FUNCTION_BLOCK AOI_LoadWoodBunk
VAR_INPUT
	execute : BOOL;
END_VAR
VAR_IN_OUT CONSTANT
	sectionID : SectionEnum;
END_VAR
VAR_IN_OUT
	robot : RobotA21;
	table : StagingTable;
	suctions : ARRAY[*] OF SuctionPad;
	//if assigned using . operator instead of (), this becomes a pointer - use numPads isntead of UPPER_BOUND/LOWER_BOUND
	loadedMaterials : ARRAY[*] OF STRING;
END_VAR
VAR_INPUT
	surfaceID : Surface;
	material : STRING;
	
	//suctionI1 : DINT;
	//suctionI2 : DINT;
	
	numPads : DINT;
END_VAR
VAR_OUTPUT
	busy : BOOL;
	done : BOOL;
	error : BOOL;
	
	recovery : BOOL;
	failCounter : INT;
	
	donePulse : BOOL;
END_VAR
VAR
	run : BOOL;
	trigger : R_TRIG;
	doneTrigger : R_TRIG;
	
	slot : INT;
	
	suctionTimer : TON;
	step : (IDLE, PREP_ROBOT, GET_FROM_TABLE, LOAD_TO_INSERTION, COMPLETE, RECOVERY_IDLE, RECOVERY_REMOVE, RECOVERY_STAGE);
END_VAR
VAR
	start, end : DINT;
	i : DINT;
	test : BOOL;
END_VAR
VAR_STAT CONSTANT
	suctionDelay : TIME := T#2S;
	suctionDistance : INT := 10;
END_VAR

{warning disable C0371}
(*
IF suctions <> 0 THEN
	FOR i:=0 TO numPads-1 BY 1 DO
		suctions[i].enable := test;
	END_FOR
END_IF
*)
trigger(CLK:= execute, Q=> );
doneTrigger(CLK:= done, Q=> donePulse);
busy := trigger.Q OR step > 0;

IF step > IDLE AND_THEN NOT preExecution() THEN //conditions to track before execution
	RETURN;
END_IF

(*
if required bunk was not found on table - restage entire table
if bunk was not loaded correctly - remove bunk, then restage entire table
*)

start := LOWER_BOUND(loadedMaterials, 1);
end := UPPER_BOUND(loadedMaterials, 1);

CASE step OF
	IDLE:
		IF trigger.Q THEN //reset outputs
			done := FALSE;
			error := FALSE;
			recovery := FALSE;
			
			step := PREP_ROBOT;
		END_IF
		
	PREP_ROBOT:
		robot.clearCommand();
		IF robot.Ready THEN
			step := GET_FROM_TABLE;
			slot := 0;
		END_IF
		
	GET_FROM_TABLE:		
		IF slot < 1 AND_THEN NOT table.findSlot(material := material, index => slot) THEN
			step := RECOVERY_STAGE;
			RETURN;
		END_IF
		
		IF NOT table.isOccupied(i := slot) AND table.getSlot(i := slot) <> '' THEN //move from table to robot gripper
			robot.HoldMaterial := table.getSlot(i := slot);
			table.remove(i := slot, material => );
		END_IF
		
		IF robot.Done THEN
			step := COMPLETE;
			RETURN;
		ELSIF robot.materialAtHoldingPosition >= 1 AND robot.materialAtHoldingPosition <= 8 THEN
			step := LOAD_TO_INSERTION;
			RETURN;
		END_IF
		
		CASE surfaceID OF
			Surface.TOP: 					robot.setGroup(group := 1, value := A21.LOAD_BUNK_TOP); 
			Surface.LEFT, Surface.RIGHT: 	robot.setGroup(group := 1, value := A21.LOAD_BUNK_SIDE);
			Surface.BOTTOM: 				robot.setGroup(group := 1, value := A21.LOAD_BUNK_BOTTOM);
		END_CASE
		robot.setGroup(group := 2, value := slot); 
			
	LOAD_TO_INSERTION:
		IF robot.materialAtHoldingPosition > 0 AND robot.HoldMaterial <> '' THEN //move from gripper to insertion
			IF loadedMaterials[surfaceID] = '' THEN //transfer to insertion as is
				loadedMaterials[surfaceID] := robot.HoldMaterial;
			ELSE //join with existing material using underscore _
				loadedMaterials[surfaceID] := JoinStrings(loadedMaterials[surfaceID], robot.HoldMaterial, '_');
			END_IF
			robot.HoldMaterial := '';
		END_IF
		
		CASE surfaceID OF
			Surface.TOP, Surface.BOTTOM:	SetSuctionsPtrArr(suctions := suctions, numPads := numPads, state := TRUE);
			Surface.LEFT, Surface.RIGHT:	SetSuctionsPtrArr(suctions := suctions, numPads := numPads, state := TRUE);
		END_CASE
		
		IF robot.Done THEN
			suctionTimer.IN := FALSE;
			step := COMPLETE;
			RETURN;
		END_IF
		
		suctionTimer(IN:= , PT:= suctionDelay, Q=> , ET=> );
		suctionTimer.IN := TRUE;
		
		IF suctionTimer.Q THEN
			robot.setGroup(group := 9, value := robot.materialAtHoldingPosition);
		END_IF
	
	COMPLETE:
		robot.clearCommand();
		
		//check insertion quality
		IF InsertionQuality(suctions := suctions, insertionMaterial := loadedMaterials[surfaceID], recipeMaterial := material) THEN
			done := TRUE;
			slot := 0;
			step := 0;
		ELSE //recovery - restage table
			failCounter := failCounter + 1;
			step := RECOVERY_IDLE;
		END_IF
		
	//---------RECOVERY-----------------------------------------
	RECOVERY_IDLE:
		robot.clearCommand();
		IF robot.Ready THEN
			step := RECOVERY_REMOVE;
		END_IF
		
	RECOVERY_REMOVE:
		IF robot.Done THEN
			step := RECOVERY_STAGE;
			RETURN;
		END_IF
		
		CASE surfaceID OF
			Surface.TOP:					robot.setGroup(group := 1, value := A21.REMOVE_BUNK_TOP);
			Surface.LEFT, Surface.RIGHT:	robot.setGroup(group := 1, value := A21.REMOVE_BUNK_SIDE);
			Surface.BOTTOM:					robot.setGroup(group := 1, value := A21.REMOVE_BUNK_BOTTOM);
		END_CASE
	
	RECOVERY_STAGE:	
		recovery := TRUE;
		error := TRUE;
		
END_CASE

METHOD PRIVATE preExecution : BOOL
VAR_INPUT
END_VAR
{warning disable C0371}
IF material = '' THEN
	done := TRUE;
	RETURN;
END_IF

IF //robot must be ready before execution
	robot.error OR 
	robot.reservation <> sectionID OR 
	robot.tool <> sectionID
THEN
	error := TRUE;
	RETURN;
END_IF

preExecution := TRUE;
END_METHOD

METHOD reset : BOOL
VAR_INPUT
END_VAR
VAR
	temp : AOI_LoadWoodBunk;
END_VAR
//(*
done := FALSE;
error := FALSE;
recovery := FALSE;
slot := 0;
step := 0;

failCounter := 0;
//*)
//THIS^ := temp;
END_METHOD

END_FUNCTION_BLOCK

(* stored: Version 1.1.0.1, ProductVersion 3.1.4024.11
   POU AOI_LoadWoodBunk: Id {8729b1eb-ce03-40b7-afa3-0137a80b10ea}, SpecialFunc None
   Method preExecution: Id {43448065-061a-4cf6-b3d1-14a86dcbddac}
   Method reset: Id {96c98ec7-6d60-41a1-9033-e9fabde425fb} *)
